DATA_BLOCK "KeyenceSR1000Ctrl_803A1DB"
{ S7_Optimized_Access := 'FALSE' }
VERSION : 0.1
NON_RETAIN
"KeyenceSR1000Ctrl"

BEGIN

END_DATA_BLOCK

